FUNCTION_BLOCK ORDER_DATA_STORAGE (* Composite Function Block Type *)
  (* Standard: 61499-2 *)
  (* Version 0.0, 12/17/2022, Dmitrii, Flexbridge AB, template *)
  PACKAGE UAO.Hackathon;
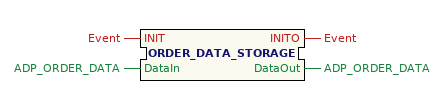
  EVENT_INPUT
    INIT;
  END_EVENT
  EVENT_OUTPUT
    INITO;
  END_EVENT
  SOCKETS
    DataIn : ADP_ORDER_DATA;
  END_SOCKETS
  PLUGS
    DataOut : ADP_ORDER_DATA;
  END_PLUGS
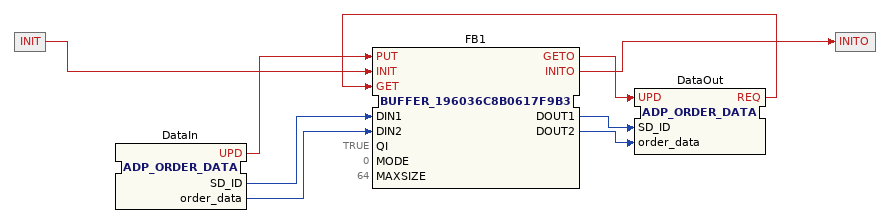
  (* TODO Replace with correct data format and storage implementation *)
  FBS
    FB1 : BUFFER_196036C8B0617F9B3(QI := TRUE, MODE := 0, MAXSIZE := 64); {SET_ATTRIBUTE(Configuration.GenericFBType.InterfaceParams, Runtime.Standard#CNT:=2;DIN${CNT$}:STRING(64),STRING(64))}
  END_FBS
  EVENT_CONNECTIONS
    DataIn.UPD TO FB1.PUT;
    INIT TO FB1.INIT;
    DataOut.REQ TO FB1.GET;
    FB1.GETO TO DataOut.UPD;
    FB1.INITO TO INITO;
  END_CONNECTIONS
  DATA_CONNECTIONS
    DataIn.SD_ID TO FB1.DIN1;
    DataIn.order_data TO FB1.DIN2;
    FB1.DOUT1 TO DataOut.SD_ID;
    FB1.DOUT2 TO DataOut.order_data;
  END_CONNECTIONS
END_FUNCTION_BLOCK
